// TIA Portal V19 export
TYPE "TetraPakV50_9_UDTNest"
   STRUCT
      OP : "OP_Int";
      Commands : "IF_Commands";
      "IF" : "TetraPakV50_9_Params";
   END_STRUCT;
END_TYPE
